// Mitsubishi GX Works2 project: servo6+   PLC: Q03UDV

PROGRAM SERVO
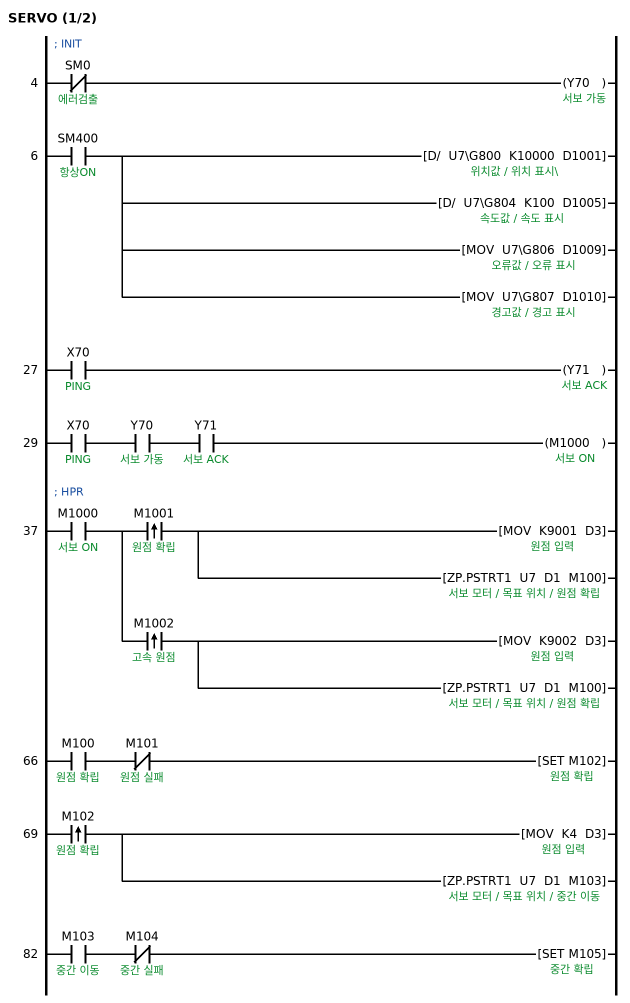
; INIT
4     LDI     SM0  ; 에러검출
      OUT     Y70  ; 서보 가동
6     LD      SM400  ; 항상ON
      D/      U7\G800 K10000 D1001  ; 위치값 / 위치 표시\
      D/      U7\G804 K100 D1005  ; 속도값 / 속도 표시
      MOV     U7\G806 D1009  ; 오류값 / 오류 표시
      MOV     U7\G807 D1010  ; 경고값 / 경고 표시
27    LD      X70  ; PING
      OUT     Y71  ; 서보 ACK
29    LD      X70  ; PING
      AND     Y70  ; 서보 가동
      AND     Y71  ; 서보 ACK
      OUT     M1000  ; 서보 ON
; HPR
37    LD      M1000  ; 서보 ON
      MPS
      ANDP    M1001  ; 원점 확립
      MOV     K9001 D3  ; 원점 입력
      ZP.PSTRT1 U7 D1 M100  ; 서보 모터 / 목표 위치 / 원점 확립
      MPP
      ANDP    M1002  ; 고속 원점
      MOV     K9002 D3
      ZP.PSTRT1 U7 D1 M100
66    LD      M100  ; 원점 확립
      ANI     M101  ; 원점 실패
      SET     M102  ; 원점 확립
69    LDP     M102  ; 원점 확립
      MOV     K4 D3
      ZP.PSTRT1 U7 D1 M103  ; 중간 이동
82    LD      M103  ; 중간 이동
      ANI     M104  ; 중간 실패
      SET     M105  ; 중간 확립
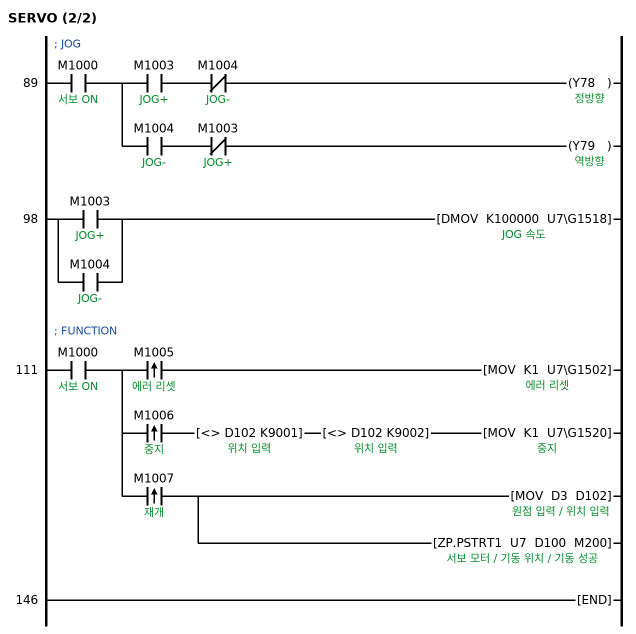
; JOG
89    LD      M1000  ; 서보 ON
      MPS
      AND     M1003  ; JOG+
      ANI     M1004  ; JOG-
      OUT     Y78  ; 정방향
      MPP
      AND     M1004  ; JOG-
      ANI     M1003  ; JOG+
      OUT     Y79  ; 역방향
98    LD      M1003  ; JOG+
      OR      M1004  ; JOG-
      DMOV    K100000 U7\G1518  ; JOG 속도
; FUNCTION
111   LD      M1000  ; 서보 ON
      MPS
      ANDP    M1005  ; 에러 리셋
      MOV     K1 U7\G1502  ; 에러 리셋
      MRD
      ANDP    M1006  ; 중지
      AND<>   D102 K9001  ; 위치 입력
      AND<>   D102 K9002  ; 위치 입력
      MOV     K1 U7\G1520  ; 중지
      MPP
      ANDP    M1007  ; 재개
      MOV     D3 D102
      ZP.PSTRT1 U7 D100 M200  ; 기동 위치 / 기동 성공
146   END
END_PROGRAM

PROGRAM MAIN
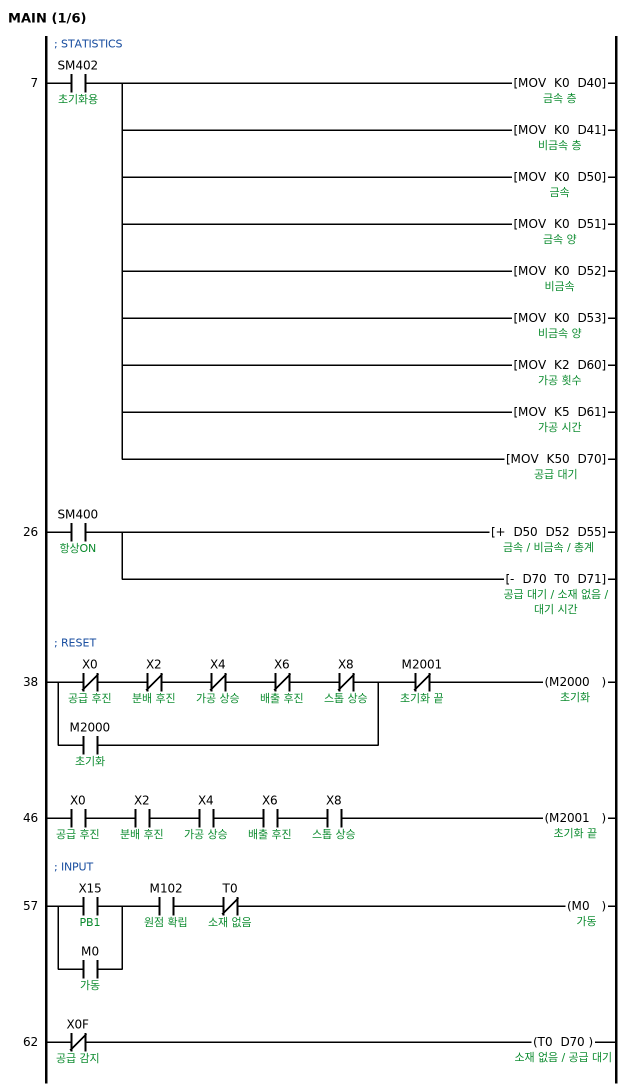
; STATISTICS
7     LD      SM402  ; 초기화용
      MOV     K0 D40  ; 금속 층
      MOV     K0 D41  ; 비금속 층
      MOV     K0 D50  ; 금속
      MOV     K0 D51  ; 금속 양
      MOV     K0 D52  ; 비금속
      MOV     K0 D53  ; 비금속 양
      MOV     K2 D60  ; 가공 횟수
      MOV     K5 D61  ; 가공 시간
      MOV     K50 D70  ; 공급 대기
26    LD      SM400  ; 항상ON
      +       D50 D52 D55  ; 총계
      -       D70 T0 D71  ; 소재 없음 / 대기 시간
; RESET
38    LDI     X0  ; 공급 후진
      ANI     X2  ; 분배 후진
      ANI     X4  ; 가공 상승
      ANI     X6  ; 배출 후진
      ANI     X8  ; 스톱 상승
      OR      M2000  ; 초기화
      ANI     M2001  ; 초기화 끝
      OUT     M2000  ; 초기화
46    LD      X0  ; 공급 후진
      AND     X2  ; 분배 후진
      AND     X4  ; 가공 상승
      AND     X6  ; 배출 후진
      AND     X8  ; 스톱 상승
      OUT     M2001  ; 초기화 끝
; INPUT
57    LD      X15  ; PB1
      OR      M0  ; 가동
      AND     M102  ; 원점 확립
      ANI     T0  ; 소재 없음
      OUT     M0  ; 가동
62    LDI     X0F  ; 공급 감지
      OUT     T0 D70  ; 소재 없음 / 공급 대기
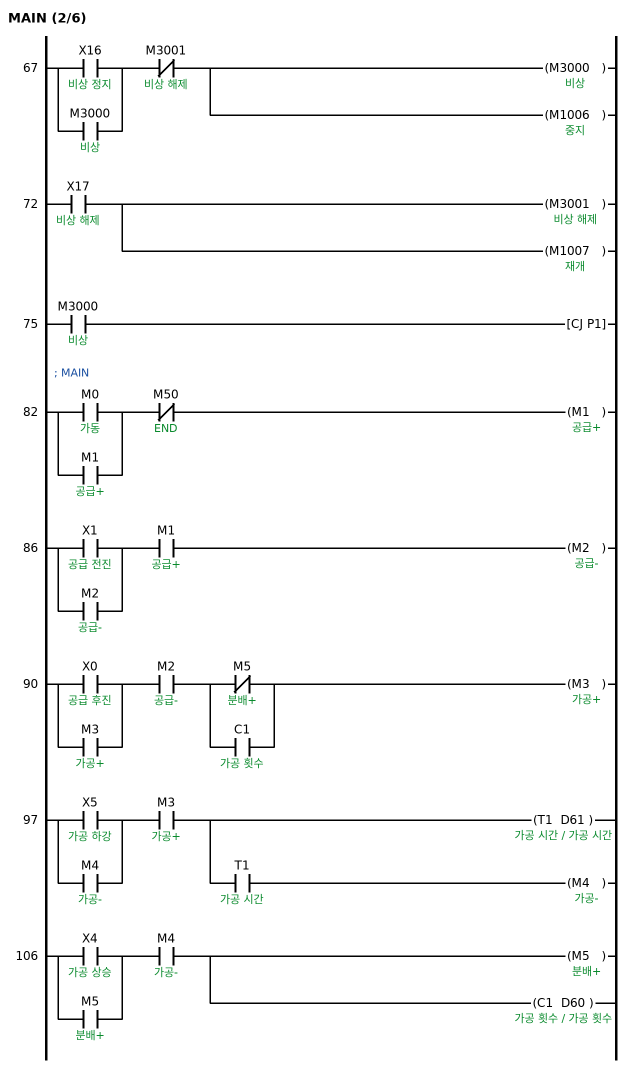
67    LD      X16  ; 비상 정지
      OR      M3000  ; 비상
      ANI     M3001  ; 비상 해제
      OUT     M3000  ; 비상
      OUT     M1006  ; 중지
72    LD      X17  ; 비상 해제
      OUT     M3001  ; 비상 해제
      OUT     M1007  ; 재개
75    LD      M3000  ; 비상
      CJ      P1  ; OUTPUT
; MAIN
82    LD      M0  ; 가동
      OR      M1  ; 공급+
      ANI     M50  ; END
      OUT     M1  ; 공급+
86    LD      X1  ; 공급 전진
      OR      M2  ; 공급-
      AND     M1  ; 공급+
      OUT     M2  ; 공급-
90    LD      X0  ; 공급 후진
      OR      M3  ; 가공+
      AND     M2  ; 공급-
      LDI     M5  ; 분배+
      OR      C1  ; 가공 횟수
      ANB
      OUT     M3  ; 가공+
97    LD      X5  ; 가공 하강
      OR      M4  ; 가공-
      AND     M3  ; 가공+
      OUT     T1 D61  ; 가공 시간 / 가공 시간
      AND     T1  ; 가공 시간
      OUT     M4  ; 가공-
106   LD      X4  ; 가공 상승
      OR      M5  ; 분배+
      AND     M4  ; 가공-
      OUT     M5  ; 분배+
      OUT     C1 D60  ; 가공 횟수 / 가공 횟수
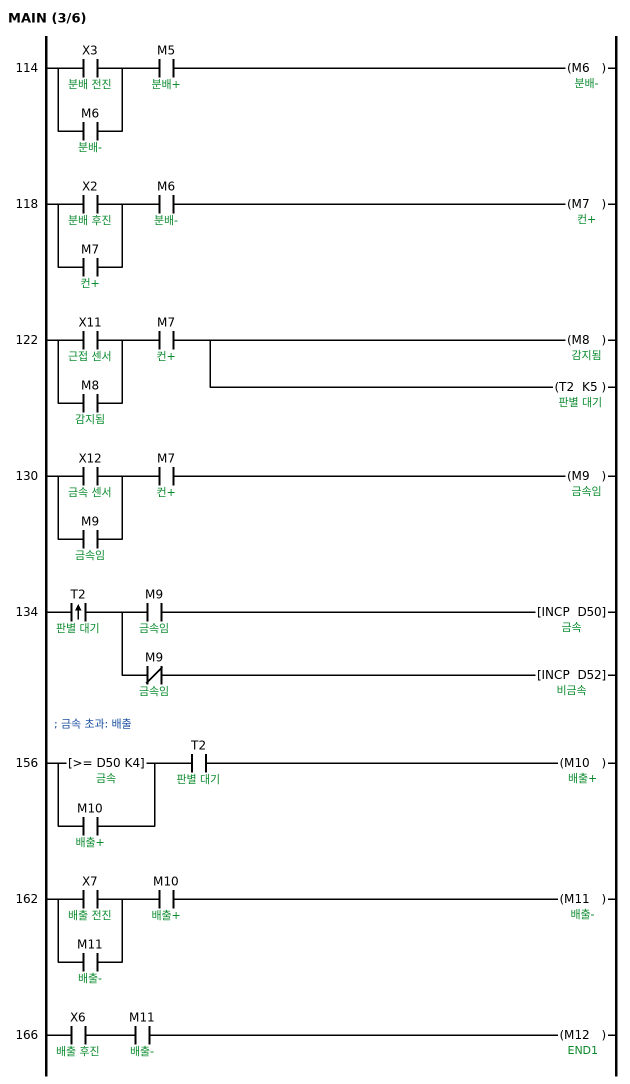
114   LD      X3  ; 분배 전진
      OR      M6  ; 분배-
      AND     M5  ; 분배+
      OUT     M6  ; 분배-
118   LD      X2  ; 분배 후진
      OR      M7  ; 컨+
      AND     M6  ; 분배-
      OUT     M7  ; 컨+
122   LD      X11  ; 근접 센서
      OR      M8  ; 감지됨
      AND     M7  ; 컨+
      OUT     M8  ; 감지됨
      OUT     T2 K5  ; 판별 대기
130   LD      X12  ; 금속 센서
      OR      M9  ; 금속임
      AND     M7  ; 컨+
      OUT     M9  ; 금속임
134   LDP     T2  ; 판별 대기
      MPS
      AND     M9  ; 금속임
      INCP    D50
      MPP
      ANI     M9  ; 금속임
      INCP    D52
; 금속 초과: 배출
156   LD>=    D50 K4  ; 금속
      OR      M10  ; 배출+
      AND     T2  ; 판별 대기
      OUT     M10  ; 배출+
162   LD      X7  ; 배출 전진
      OR      M11  ; 배출-
      AND     M10  ; 배출+
      OUT     M11  ; 배출-
166   LD      X6  ; 배출 후진
      AND     M11  ; 배출-
      OUT     M12  ; END1
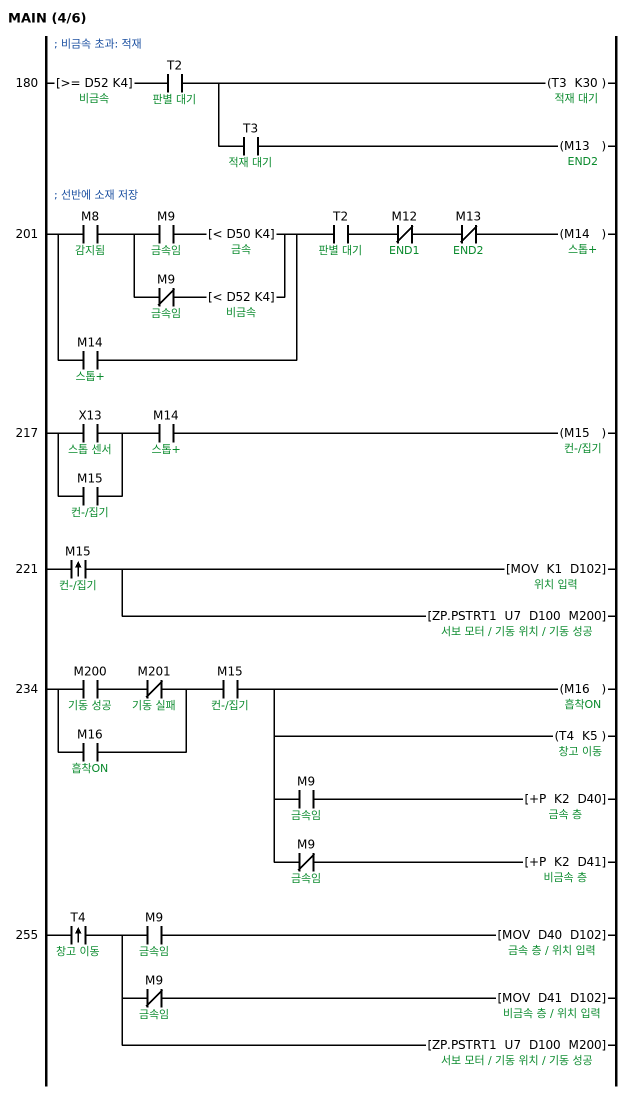
; 비금속 초과: 적재
180   LD>=    D52 K4  ; 비금속
      AND     T2  ; 판별 대기
      OUT     T3 K30  ; 적재 대기
      AND     T3  ; 적재 대기
      OUT     M13  ; END2
; 선반에 소재 저장
201   LD      M8  ; 감지됨
      LD      M9  ; 금속임
      AND<    D50 K4  ; 금속
      LDI     M9  ; 금속임
      AND<    D52 K4  ; 비금속
      ORB
      ANB
      OR      M14  ; 스톱+
      AND     T2  ; 판별 대기
      ANI     M12  ; END1
      ANI     M13  ; END2
      OUT     M14  ; 스톱+
217   LD      X13  ; 스톱 센서
      OR      M15  ; 컨-/집기
      AND     M14  ; 스톱+
      OUT     M15  ; 컨-/집기
221   LDP     M15  ; 컨-/집기
      MOV     K1 D102  ; 위치 입력
      ZP.PSTRT1 U7 D100 M200  ; 서보 모터 / 기동 위치 / 기동 성공
234   LD      M200  ; 기동 성공
      ANI     M201  ; 기동 실패
      OR      M16  ; 흡착ON
      AND     M15  ; 컨-/집기
      OUT     M16  ; 흡착ON
      OUT     T4 K5  ; 창고 이동
      MPS
      AND     M9  ; 금속임
      +P      K2 D40
      MPP
      ANI     M9  ; 금속임
      +P      K2 D41
255   LDP     T4  ; 창고 이동
      MPS
      AND     M9  ; 금속임
      MOV     D40 D102
      MRD
      ANI     M9  ; 금속임
      MOV     D41 D102
      MPP
      ZP.PSTRT1 U7 D100 M200
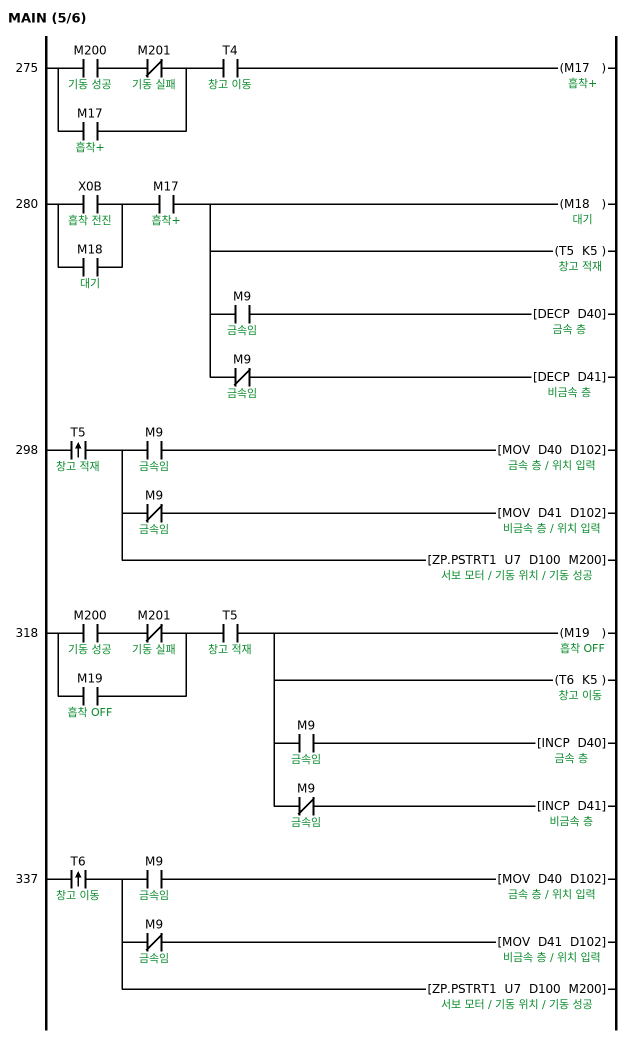
275   LD      M200  ; 기동 성공
      ANI     M201  ; 기동 실패
      OR      M17  ; 흡착+
      AND     T4  ; 창고 이동
      OUT     M17  ; 흡착+
280   LD      X0B  ; 흡착 전진
      OR      M18  ; 대기
      AND     M17  ; 흡착+
      OUT     M18  ; 대기
      OUT     T5 K5  ; 창고 적재
      MPS
      AND     M9  ; 금속임
      DECP    D40
      MPP
      ANI     M9  ; 금속임
      DECP    D41
298   LDP     T5  ; 창고 적재
      MPS
      AND     M9  ; 금속임
      MOV     D40 D102
      MRD
      ANI     M9  ; 금속임
      MOV     D41 D102
      MPP
      ZP.PSTRT1 U7 D100 M200
318   LD      M200  ; 기동 성공
      ANI     M201  ; 기동 실패
      OR      M19  ; 흡착 OFF
      AND     T5  ; 창고 적재
      OUT     M19  ; 흡착 OFF
      OUT     T6 K5  ; 창고 이동
      MPS
      AND     M9  ; 금속임
      INCP    D40
      MPP
      ANI     M9  ; 금속임
      INCP    D41
337   LDP     T6  ; 창고 이동
      MPS
      AND     M9  ; 금속임
      MOV     D40 D102
      MRD
      ANI     M9  ; 금속임
      MOV     D41 D102
      MPP
      ZP.PSTRT1 U7 D100 M200
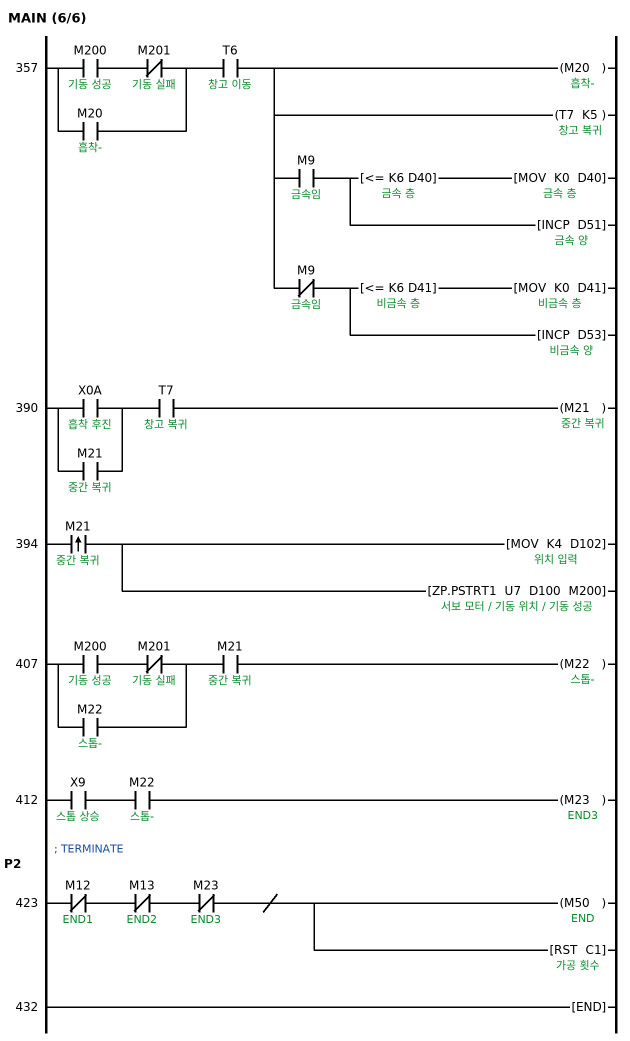
357   LD      M200  ; 기동 성공
      ANI     M201  ; 기동 실패
      OR      M20  ; 흡착-
      AND     T6  ; 창고 이동
      OUT     M20  ; 흡착-
      OUT     T7 K5  ; 창고 복귀
      MPS
      AND     M9  ; 금속임
      MPS
      AND<=   K6 D40  ; 금속 층
      MOV     K0 D40
      MPP
      INCP    D51
      MPP
      ANI     M9  ; 금속임
      MPS
      AND<=   K6 D41  ; 비금속 층
      MOV     K0 D41
      MPP
      INCP    D53
390   LD      X0A  ; 흡착 후진
      OR      M21  ; 중간 복귀
      AND     T7  ; 창고 복귀
      OUT     M21  ; 중간 복귀
394   LDP     M21  ; 중간 복귀
      MOV     K4 D102
      ZP.PSTRT1 U7 D100 M200
407   LD      M200  ; 기동 성공
      ANI     M201  ; 기동 실패
      OR      M22  ; 스톱-
      AND     M21  ; 중간 복귀
      OUT     M22  ; 스톱-
412   LD      X9  ; 스톱 상승
      AND     M22  ; 스톱-
      OUT     M23  ; END3
; TERMINATE
      P2
423   LDI     M12  ; END1
      ANI     M13  ; END2
      ANI     M23  ; END3
      INV
      OUT     M50  ; END
      RST     C1  ; 가공 횟수
432   END
END_PROGRAM

PROGRAM OUTPUT
; OUTPUT
      P1
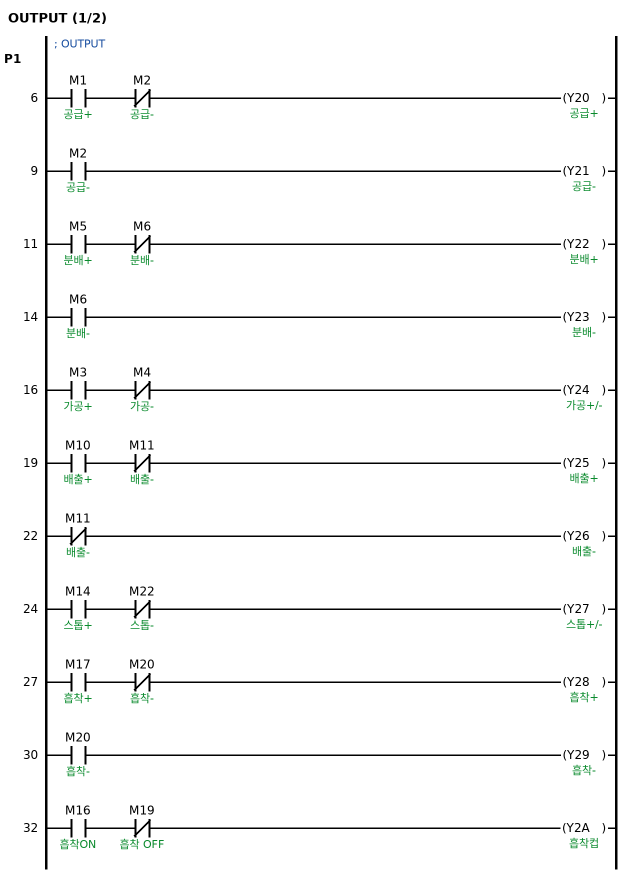
6     LD      M1  ; 공급+
      ANI     M2  ; 공급-
      OUT     Y20  ; 공급+
9     LD      M2  ; 공급-
      OUT     Y21  ; 공급-
11    LD      M5  ; 분배+
      ANI     M6  ; 분배-
      OUT     Y22  ; 분배+
14    LD      M6  ; 분배-
      OUT     Y23  ; 분배-
16    LD      M3  ; 가공+
      ANI     M4  ; 가공-
      OUT     Y24  ; 가공+/-
19    LD      M10  ; 배출+
      ANI     M11  ; 배출-
      OUT     Y25  ; 배출+
22    LDI     M11  ; 배출-
      OUT     Y26  ; 배출-
24    LD      M14  ; 스톱+
      ANI     M22  ; 스톱-
      OUT     Y27  ; 스톱+/-
27    LD      M17  ; 흡착+
      ANI     M20  ; 흡착-
      OUT     Y28  ; 흡착+
30    LD      M20  ; 흡착-
      OUT     Y29  ; 흡착-
32    LD      M16  ; 흡착ON
      ANI     M19  ; 흡착 OFF
      OUT     Y2A  ; 흡착컵
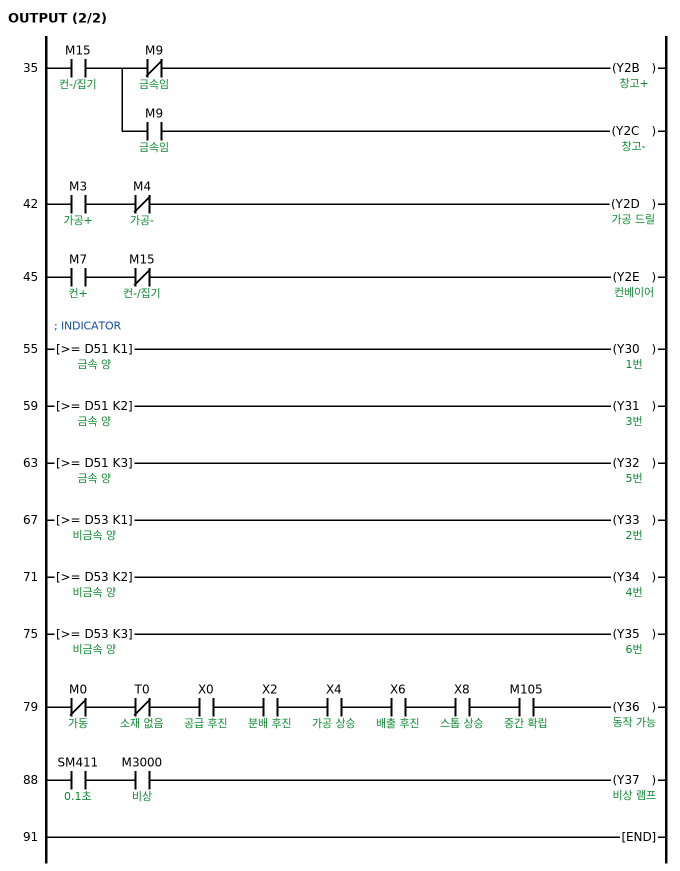
35    LD      M15  ; 컨-/집기
      MPS
      ANI     M9  ; 금속임
      OUT     Y2B  ; 창고+
      MPP
      AND     M9  ; 금속임
      OUT     Y2C  ; 창고-
42    LD      M3  ; 가공+
      ANI     M4  ; 가공-
      OUT     Y2D  ; 가공 드릴
45    LD      M7  ; 컨+
      ANI     M15  ; 컨-/집기
      OUT     Y2E  ; 컨베이어
; INDICATOR
55    LD>=    D51 K1  ; 금속 양
      OUT     Y30  ; 1번
59    LD>=    D51 K2  ; 금속 양
      OUT     Y31  ; 3번
63    LD>=    D51 K3  ; 금속 양
      OUT     Y32  ; 5번
67    LD>=    D53 K1  ; 비금속 양
      OUT     Y33  ; 2번
71    LD>=    D53 K2  ; 비금속 양
      OUT     Y34  ; 4번
75    LD>=    D53 K3  ; 비금속 양
      OUT     Y35  ; 6번
79    LDI     M0  ; 가동
      ANI     T0  ; 소재 없음
      AND     X0  ; 공급 후진
      AND     X2  ; 분배 후진
      AND     X4  ; 가공 상승
      AND     X6  ; 배출 후진
      AND     X8  ; 스톱 상승
      AND     M105  ; 중간 확립
      OUT     Y36  ; 동작 가능
88    LD      SM411  ; 0.1초
      AND     M3000  ; 비상
      OUT     Y37  ; 비상 램프
91    END
END_PROGRAM

// device comments not shown above
X0C  ; 흡착 후진
X0D  ; 창고 전진
X0E  ; 창고 후진
Y40  ; 원점 램프
Y41  ; 원점 확립
Y42  ; 비상등
D30  ; 층 수
T8  ; 복귀 대기
P2  ; END
